{attribute addProperty BoxType "EJ2914-0000-0017"}
{attribute addProperty Id "FSoE_InputsFSoE_Inputs_74C0DA41486FSoE_OutputsFSoE_Outputs_841EDA4B486"}
{attribute addProperty CRC "3516287219"}
{attribute addProperty SizeInBites "96"}
{attribute addProperty SizeInBytes "12"}
TYPE Module_1_FSOE_D19648F3 :
STRUCT
	{attribute addProperty Name "FSoE_Inputs"}
	FSoE_Inputs  : FSoE_Inputs_74C0DA41;
	{attribute addProperty Name "FSoE_Outputs"}
	FSoE_Outputs  : FSoE_Outputs_841EDA4B;
END_STRUCT
END_TYPE

(* stored: Version 1.2.0.0, ProductVersion 3.1.4024.9
   DUT Module_1_FSOE_D19648F3: Id {df03cfb1-a81b-470a-9149-054e8bada2ec} *)
